Universal Robots URScript: Fase5.script

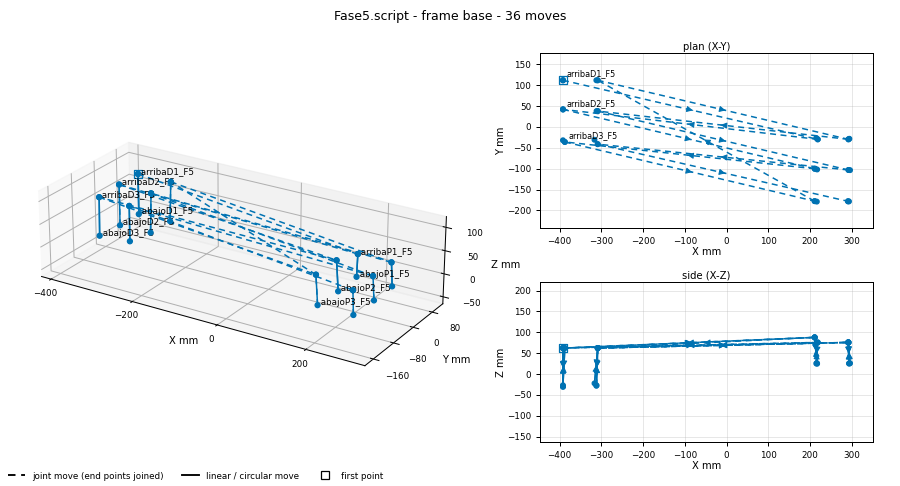
[picture p0: tool path of Fase5.script in frame base, 36 of 39 moves have a stored position in this frame; points joined in program order, loops and branches not executed]
def Fase5():
  step_count_3c5ae5f3_6041_43ff_bf36_90ec5d0922ff = 0.0
  thread Step_Counter_Thread_5067f2b5_ec87_46cd_b1bd_ecc09904e503():
    while (True):
      step_count_3c5ae5f3_6041_43ff_bf36_90ec5d0922ff = step_count_3c5ae5f3_6041_43ff_bf36_90ec5d0922ff + 1.0
      sync()
    end
  end
  run Step_Counter_Thread_5067f2b5_ec87_46cd_b1bd_ecc09904e503()
  set_standard_analog_input_domain(0, 1)
  set_standard_analog_input_domain(1, 1)
  set_tool_analog_input_domain(0, 1)
  set_tool_analog_input_domain(1, 1)
  set_analog_outputdomain(0, 0)
  set_analog_outputdomain(1, 0)
  set_input_actions_to_default()
  set_tool_communication(True, 1000000, 2, 1, 1.5, 3.5)
  set_tool_output_mode(0)
  set_tool_digital_output_mode(0, 1)
  set_tool_digital_output_mode(1, 1)
  set_tool_voltage(0)
  set_gravity([0.0, 0.0, 9.82])
  set_safety_mode_transition_hardness(1)
  set_tcp(p[0.00755148296704608,0.003639298738154023,0.026409592411711,0.0,0.0,0.0])
  set_payload(1.14, [0.022, -0.007, 0.054])
  global Mesa=p[-0.3283222416297581,-0.20095078680444134,-0.01154506462095492,-2.1087277613487028,-2.3273776320839428,-7.166709239352482E-4]
  # begin: URCap Installation Node
  #   Source: Remote TCP & Toolpath, 1.2.65.build36, Universal Robots A/S
  #   Type: Remote TCP & Toolpath
  # end: URCap Installation Node
  # begin: URCap Installation Node
  #   Source: OnRobot, 5.1.6, OnRobot A/S
  #   Type: Configuración de OnRobot
  on_robot_type = 3
  on_robot_cycle = 2.0
  on_device_ip = "localhost"
  on_device_socket_port = 51234
  on_xmlrpc = rpc_factory("xmlrpc", "http://localhost:41414")
  on_RPC = rpc_factory("xmlrpc", "http://127.0.0.1:31416")
  ON_DEBUG_LOG = False
  on_isMetric = True
  on_toolConnector = True
  on_ioqc = False
  on_dual = False
  on_ft = False
  on_hex = False
  on_gecko = 0
  on_gripper = [False, False, False]
  #======    OnRobot Globals    ======#

  ON_MATH_PI=3.141593
  ON_ZEROPOSE=p[0.0,0.0,0.0,0.0,0.0,0.0]
  ON_ZEROFRAME=p[0.0,0.0,0.0,0.0,0.0,0.0]
  ON_ZERO3D=[0.0,0.0,0.0]
  ON_ZERO6D=[0.0,0.0,0.0,0.0,0.0,0.0]
  ON_ZERO8D=[0.0,0.0,0.0,0.0,0.0,0.0,0.0,0.0]
  ON_FALSE3D=[False,False,False]
  ON_FALSE6D=[False,False,False,False,False,False]
  ON_FALSE8D=[False,False,False,False,False,False,False,False]
  global on_return=0
  on_speedL=ON_ZERO6D
  on_speedBase=ON_ZERO6D
  on_speedVect=ON_ZERO6D
  on_speedExtra=ON_ZERO6D
  on_speedDC=ON_ZERO6D
  on_speedGecko=ON_ZERO6D
  on_floatRegShift=24
  on_intRegShift=24
  on_boolRegShift=64
  ON_BASE_SHIFT_FLOAT=24
  ON_BASE_SHIFT_INT=24
  ON_BASE_SHIFT_BOOL=64
  ON_DEVICE_SHIFT_FLOAT=3
  ON_DEVICE_SHIFT_INT=2
  ON_DEVICE_SHIFT_BOOL=7
  ON_COMMON_SHIFT_FLOAT=12
  ON_COMMON_SHIFT_INT=3
  ON_COMMON_SHIFT_BOOL=1
  ON_DI_SINGLE=0
  ON_DI_PRIMARY=1
  ON_DI_SECONDARY=2
  ON_DI_DUAL=3
  ON_DEVICE_ID_MISSING=0
  ON_INIT_TIMEOUT=500
  on_robot_TCP_offset=ON_ZEROFRAME
  on_tcp_offset_actual=ON_ZEROFRAME
  on_cog_actual=ON_ZEROFRAME
  on_mass_actual=0.0
  on_robot_mount=[0.0,0.0]

  #======    End of OnRobot Globals    ======#
  #======    OnRobot Interface Messages    ======#

  on_devices_primary_log="Dispositivos de OnRobot"
  on_devices_secondary_log="Dispositivo secundario de OnRobot"
  on_device_error_title="OnRobot - Error de dispositivo"
  on_install_error="La configuración de OnRobot no es correcta.<br>Compruebe el estado en la página de configuración de OnRobot, en la pestaña de instalación.<br>Programa detenido."
  on_device_missing="No hay ningún dispositivo conectado.<br>Programa detenido."
  ft_device_missing="No hay ningún sensor F/T OnRobot conectado.<br>Programa detenido."
  rg2ft_device_missing="No hay ninguna pinza RG2-FT conectada.<br>Programa detenido."
  rg_device_missing="No hay ninguna pinza RG conectada.<br>Programa detenido."
  vg_device_missing="No hay ninguna pinza VG conectada.<br>Programa detenido."
  gg_device_missing="No hay ninguna Gecko Gripper conectada.<br>Programa detenido."
  sg_device_missing="No hay ninguna Soft Gripper conectada.<br>Programa detenido."
  tfg_device_missing="No hay ninguna pinza 3FG conectada.<br>Programa detenido."
  on_xmlrpc_start_ip="Conexión al servidor XML-RPC de OnRobot:"
  on_java_comm_error_textmsg_title="OnRobot - Error de comunicación:"
  on_java_comm_controlsocket_open_error="Apertura de la toma 'javaSocket' incorrecta."
  on_java_comm_error_title="OnRobot - Error de comunicación"
  on_java_comm_socket_open_error="El establecimiento de la conexión con el URCap ha excedido el tiempo.<br>Compruebe el estado en la página de configuración de OnRobot, en la pestaña de instalación.<br>Programa detenido."
  on_rtde_feed_error_textmsg_title="OnRobot - Error de comunicación:"
  on_rtde_feed_open_error_textmsg="Apertura de la toma 'rtdeFeed' incorrecta."
  on_rtde_feed_error_title="OnRobot - Error de comunicación"
  on_rtde_feed_open_error="El establecimiento de la conexión con los dispositivos ha excedido el tiempo.<br>Asegúrese de que los dispositivos de OnRobot funcionen y compruebe el estado en la página de configuración de OnRobot, en la pestaña de instalación."

  #======    End of OnRobot Interface Messages    ======#
  #======    OnRobot Interface    ======#

  on_portopened_javaSocket=False
  on_rtde_feed_opened=False
  on_dataRead_running=False
  FT_SENSOR_ID_UNDEFINED=0
  FT_SENSOR_ID_UNKNOWN=1
  FT_SENSOR_ID_HEX_V1=11
  FT_SENSOR_ID_HEX_V2=12
  FT_SENSOR_ID_HEX_V3=13
  FT_SENSOR_ID_RG2FT_V0=20
  FT_SENSOR_ID_RG2FT_V1=21
  FT_SENSOR_ID_RG2FT_V2=22
  def on_error(status_flag,message,title,stop_var=False):
  if(status_flag):
  popup(message,title=title,error=True,blocking=False)
  stop_var=True
  end
  return stop_var
  end
  def on_warning(status_flag,message,title):
  if(status_flag):
  textmsg(title,message)
  end
  end
  def on_missing():
  popup(on_device_missing,title=on_device_error_title,error=True,blocking=False)
  halt
  end
  def ft_missing():
  popup(ft_device_missing,title=on_device_error_title,error=True,blocking=False)
  halt
  end
  def rg2ft_missing():
  popup(rg2ft_device_missing,title=on_device_error_title,error=True,blocking=False)
  halt
  end
  def rg_missing():
  popup(rg_device_missing,title=on_device_error_title,error=True,blocking=False)
  halt
  end
  def vg_missing():
  popup(vg_device_missing,title=on_device_error_title,error=True,blocking=False)
  halt
  end
  def gg_missing():
  popup(gg_device_missing,title=on_device_error_title,error=True,blocking=False)
  halt
  end
  def sg_missing():
  popup(sg_device_missing,title=on_device_error_title,error=True,blocking=False)
  halt
  end
  def tfg_missing():
  popup(tfg_device_missing,title=on_device_error_title,error=True,blocking=False)
  halt
  end
  def on_portclose_javaSocket():
  socket_close("javaSocket")
  on_portopened_javaSocket=False
  end
  def on_portopen_javaSocket():
  on_portclose_javaSocket()
  on_portopened_javaSocket=socket_open("127.0.0.1",44005,"javaSocket")
  if not on_portopened_javaSocket:
  textmsg(on_java_comm_error_textmsg_title,on_java_comm_controlsocket_open_error)
  popup(on_java_comm_socket_open_error,title=on_java_comm_error_title,error=True,blocking=False)
  halt
  end
  end
  def on_rtde_feed_close():
  socket_close("rtdeFeed")
  on_rtde_feed_opened=False
  end
  def on_rtde_feed_open():
  on_rtde_feed_close()
  on_rtde_feed_opened=socket_open(on_device_ip,on_device_socket_port,"rtdeFeed")
  if not on_rtde_feed_opened:
  on_rtde_feed_opened=socket_open(on_device_ip,on_device_socket_port,"rtdeFeed")
  end
  if not on_rtde_feed_opened:
  textmsg(on_rtde_feed_error_textmsg_title,on_rtde_feed_open_error_textmsg)
  popup(on_rtde_feed_open_error,title=on_rtde_feed_error_title,error=True,blocking=False)
  halt
  end
  end
  def on_dataRead():
  enter_critical
  floatRegDummy=read_input_float_register(0+on_floatRegShift)
  on_speedVect[0]=floatRegDummy/1000.0
  floatRegDummy=read_input_float_register(1+on_floatRegShift)
  on_speedVect[1]=floatRegDummy/1000.0
  floatRegDummy=read_input_float_register(2+on_floatRegShift)
  on_speedVect[2]=floatRegDummy/1000.0
  floatRegDummy=read_input_float_register(3+on_floatRegShift)
  on_speedVect[3]=floatRegDummy
  floatRegDummy=read_input_float_register(4+on_floatRegShift)
  on_speedVect[4]=floatRegDummy
  floatRegDummy=read_input_float_register(5+on_floatRegShift)
  on_speedVect[5]=floatRegDummy
  exit_critical
  end
  def on_set_rtde_watchdog(updateHz=5,ftWD=False,gripperWD=-1):
  local update_str=str_cat(" watchdog set to [Hz]: ",updateHz)
  if ftWD:
  watchdog_int_reg_str=str_cat("input_int_register_",0+on_intRegShift)
  rtde_set_watchdog(watchdog_int_reg_str,updateHz,"stop")
  if ON_DEBUG_LOG:
  textmsg(watchdog_int_reg_str,update_str)
  end
  end
  if not(gripperWD<0):
  if(gripperWD==ON_DI_SINGLE or gripperWD==ON_DI_PRIMARY or gripperWD==ON_DI_DUAL):
  watchdog_int_reg_str=str_cat("input_int_register_",3+on_intRegShift)
  rtde_set_watchdog(watchdog_int_reg_str,updateHz,"stop")
  if ON_DEBUG_LOG:
  textmsg(watchdog_int_reg_str,update_str)
  end
  end
  if(gripperWD==ON_DI_SECONDARY or gripperWD==ON_DI_DUAL):
  watchdog_int_reg_str=str_cat("input_int_register_",ON_DEVICE_SHIFT_INT+3+on_intRegShift)
  rtde_set_watchdog(watchdog_int_reg_str,updateHz,"stop")
  if ON_DEBUG_LOG:
  textmsg(watchdog_int_reg_str,update_str)
  end
  end
  end
  end
  def on_speedVect_get():
  return[on_speedVect[0],on_speedVect[1],on_speedVect[2],on_speedVect[3],on_speedVect[4],on_speedVect[5]]
  end
  def on_speedDC_get():
  local speedExtra=ON_ZERO6D
  if on_speedl_for_depthcompensation:
  speedExtra=[on_speedDC[0],on_speedDC[1],on_speedDC[2],on_speedDC[3],on_speedDC[4],on_speedDC[5]]
  end
  return speedExtra
  end
  def on_speedDC_set(speedDC):
  on_speedDC=[speedDC[0],speedDC[1],speedDC[2],speedDC[3],speedDC[4],speedDC[5]]
  end
  def on_speedGecko_get():
  local speedExtra=ON_ZERO6D
  if on_speedl_for_gecko:
  speedExtra=[on_speedGecko[0],on_speedGecko[1],on_speedGecko[2],on_speedGecko[3],on_speedGecko[4],on_speedGecko[5]]
  end
  return speedExtra
  end
  def on_speedGecko_set(speedGecko):
  on_speedGecko=[speedGecko[0],speedGecko[1],speedGecko[2],speedGecko[3],speedGecko[4],speedGecko[5]]
  end
  thread on_dataRead_thread():
  if ON_DEBUG_LOG:
  textmsg("Starting on_dataRead thread")
  end
  while on_dataRead_running:
  sync()
  on_dataRead()
  end
  if ON_DEBUG_LOG:
  textmsg("Stopping on_dataRead thread")
  end
  end

  #======    End of OnRobot Interface    ======#
  #======    OnRobot QC Setup Tool Connector    ======#

  def tc_setup_tool():
  if ON_DEBUG_LOG:
  textmsg("QC Setup Tool Connector start...")
  end
  set_tool_voltage(24)

  set_tool_communication(True,1000000,2,1,1.5,3.5)

  if ON_DEBUG_LOG:
  textmsg("QC Setup Tool Connector end.")
  end
  end

  #======    End of OnRobot QC Setup Tool Connector    ======#
  #======    OnRobot TCP Messages    ======#

  on_tcp_log_msg_default="OnRobot: Desplazamiento del TCP del robot establecido en:"
  on_tcp_log_msg_primary="OnRobot: Desplazamiento del TCP del robot establecido en primario:"
  on_tcp_log_msg_secondary="OnRobot: Desplazamiento del TCP del robot establecido en secundario:"

  #======    End of OnRobot TCP Messages    ======#
  #======    OnRobot TCP    ======#

  on_tcp_offset_actual=ON_ZEROFRAME
  on_tcp_offset_primary=ON_ZEROFRAME
  on_tcp_static_primary=ON_ZEROFRAME
  on_tcp_dynamic_primary=ON_ZEROFRAME
  on_tcp_vision_primary=ON_ZEROFRAME
  on_tcp_qc_primary=ON_ZEROFRAME
  on_tcp_base_primary=ON_ZEROFRAME
  on_tcp_gripper_static_primary=ON_ZEROFRAME
  on_tcp_tool_primary=ON_ZEROFRAME
  on_tcp_gripper_dynamic_primary=ON_ZEROFRAME
  on_tcp_gripper_primary=ON_ZEROFRAME
  on_tcp_offset_secondary=ON_ZEROFRAME
  on_tcp_static_secondary=ON_ZEROFRAME
  on_tcp_dynamic_secondary=ON_ZEROFRAME
  on_tcp_vision_secondary=ON_ZEROFRAME
  on_tcp_qc_secondary=ON_ZEROFRAME
  on_tcp_base_secondary=ON_ZEROFRAME
  on_tcp_gripper_static_secondary=ON_ZEROFRAME
  on_tcp_tool_secondary=ON_ZEROFRAME
  on_tcp_gripper_dynamic_secondary=ON_ZEROFRAME
  on_tcp_gripper_secondary=ON_ZEROFRAME
  def on_tcp_update_primary():
  if ON_DEBUG_LOG:
  textmsg("TCP Update Primary start..")
  end
  on_tcp_gripper_dynamic_primary=p[0.0, 0.0, 0.0, 0.0, 0.0, 0.0]
  enter_critical
  on_tcp_dynamic_primary=pose_trans(on_tcp_static_primary,on_tcp_gripper_dynamic_primary)
  on_tcp_offset_primary=pose_trans(on_tcp_dynamic_primary,on_tcp_tool_primary)
  exit_critical
  if ON_DEBUG_LOG:
  textmsg("TCP Update Primary end.")
  end
  end
  def on_tcp_init_primary():
  if ON_DEBUG_LOG:
  textmsg("TCP Init Primary start..")
  end
  enter_critical
  on_tcp_base_primary=pose_trans(on_tcp_vision_primary,on_tcp_qc_primary)
  on_tcp_static_primary=pose_trans(on_tcp_base_primary,on_tcp_gripper_static_primary)
  exit_critical
  on_tcp_update_primary()
  if ON_DEBUG_LOG:
  textmsg("TCP Init Primary end.")
  end
  end
  def on_tcp_offset_set(TCP_offset):
  if ON_DEBUG_LOG:
  textmsg("TCP Offset set started!")
  end
  on_tcp_offset_send(TCP_offset)
  if(on_follow_tcp):
  set_tcp(TCP_offset)
  end
  on_robot_TCP_offset=TCP_offset
  if ON_DEBUG_LOG:
  textmsg("TCP Offset set to: ",on_robot_TCP_offset)
  end
  end
  def on_tcp_offset_forced_set_actual(isPrimary=True):
  if(not on_follow_tcp):

  local tcp_log_msg=on_tcp_log_msg_default

  textmsg(tcp_log_msg,on_tcp_offset_actual)
  set_tcp(on_tcp_offset_actual)
  end
  end
  def on_tcp_update(isPrimary=True):
  on_tcp_update_primary()

  on_tcp_set_actual_to(isPrimary)
  end
  def on_tcp_set_actual_to(isPrimary=True):

  on_tcp_offset_actual=on_tcp_offset_primary
  if(on_follow_tcp):
  textmsg(on_tcp_log_msg_default,on_tcp_offset_actual)
  end

  on_tcp_active_is_primary=isPrimary
  on_tcp_offset_set(on_tcp_offset_actual)
  end
  def on_tcp_update_tool_primary(tool_offset):
  if ON_DEBUG_LOG:
  textmsg("TCP Update Tool Primary start..")
  end
  on_tcp_tool_primary=tool_offset
  on_tcp_update_primary()
  if ON_DEBUG_LOG:
  textmsg("TCP Update Tool Primary end.")
  end
  end
  def on_tcp_tool_rpy_get(xyz=[0.0,0.0,0.0],rpy=[0.0,0.0,0.0]):
  local rotvec=rpy2rotvec(rpy)
  local tool_offset=p[xyz[0],xyz[1],xyz[2],rotvec[0],rotvec[1],rotvec[2]]
  return tool_offset
  end

  def on_tcp_update_tool(tool_offset,tool_index=0):
  if ON_DEBUG_LOG:
  textmsg("TCP Update Tool start..")
  end
  if(tool_index!=ON_DI_SECONDARY):
  on_tcp_update_tool_primary(tool_offset)
  local isPrimary=True

  end
  on_tcp_set_actual_to(isPrimary)
  if ON_DEBUG_LOG:
  textmsg("TCP Update Tool end.")
  end
  end

  #======    End of OnRobot TCP    ======#
  #======    OnRobot Payload Messages    ======#

  on_mass_log_msg="OnRobot: Masa de la carga útil del robot establecida en:"
  on_cog_log_msg="OnRobot: Centro de gravedad de la carga útil del robot establecido en:"

  #======    End of OnRobot Payload Messages    ======#
  #======    OnRobot Payload    ======#

  on_cog_actual=ON_ZEROFRAME
  on_mass_actual=0.0
  on_cog_primary=ON_ZEROFRAME
  on_cog_L1L2_primary=ON_ZEROFRAME
  on_mass_primary=0.0
  on_mass_L1L2_primary=0.0
  on_cog_vision_primary=ON_ZEROFRAME
  on_cog_qc_primary=ON_ZEROFRAME
  on_cog_base_primary=ON_ZEROFRAME
  on_cog_gripper_primary=ON_ZEROFRAME
  on_cog_tool_primary=ON_ZEROFRAME
  on_mass_vision_primary=0.0
  on_mass_qc_primary=0.0
  on_mass_base_primary=0.0
  on_mass_gripper_primary=0.0
  on_mass_tool_primary=0.0
  on_cog_secondary=ON_ZEROFRAME
  on_mass_secondary=0.0
  on_cog_gripper_secondary=ON_ZEROFRAME
  on_mass_gripper_secondary=0.0
  on_cog_tool_secondary=ON_ZEROFRAME
  on_mass_tool_secondary=0.0
  ON_LB2KG001=0.45359237/100
  def on_payload_update_primary():
  if ON_DEBUG_LOG:
  textmsg("Payload Update Primary start..")
  end
  enter_critical
  on_mass_primary=on_mass_L1L2_primary+on_mass_tool_primary
  local massL1L2L3Ratio=on_mass_tool_primary/on_mass_primary
  local toolAbsCOG=pose_trans(on_tcp_dynamic_primary,on_cog_tool_primary)
  toolAbsCOG=p[toolAbsCOG[0],toolAbsCOG[1],toolAbsCOG[2],0.0,0.0,0.0]
  on_cog_primary=interpolate_pose(on_cog_L1L2_primary,toolAbsCOG,massL1L2L3Ratio)
  on_cog_primary=p[on_cog_primary[0],on_cog_primary[1],on_cog_primary[2],0.0,0.0,0.0]
  exit_critical
  if ON_DEBUG_LOG:
  textmsg("Payload Update Primary end.")
  end
  end
  def on_payload_init_primary():
  if ON_DEBUG_LOG:
  textmsg("Payload Init Primary start..")
  end
  enter_critical
  on_mass_base_primary=on_mass_vision_primary+on_mass_qc_primary
  local massL0L1Ratio=on_mass_qc_primary/on_mass_base_primary
  on_mass_L1L2_primary=on_mass_base_primary+on_mass_gripper_primary
  local massL1L2Ratio=on_mass_gripper_primary/on_mass_L1L2_primary
  local qcAbsCOG=pose_trans(on_tcp_vision_primary,on_cog_qc_primary)
  qcAbsCOG=p[qcAbsCOG[0],qcAbsCOG[1],qcAbsCOG[2],0.0,0.0,0.0]
  on_cog_base_primary=interpolate_pose(on_cog_vision_primary,qcAbsCOG,massL0L1Ratio)
  on_cog_base_primary=p[on_cog_base_primary[0],on_cog_base_primary[1],on_cog_base_primary[2],0.0,0.0,0.0]
  local gripperAbsCOG=pose_trans(on_tcp_base_primary,on_cog_gripper_primary)
  gripperAbsCOG=p[gripperAbsCOG[0],gripperAbsCOG[1],gripperAbsCOG[2],0.0,0.0,0.0]
  on_cog_L1L2_primary=interpolate_pose(on_cog_base_primary,gripperAbsCOG,massL1L2Ratio)
  on_cog_L1L2_primary=p[on_cog_L1L2_primary[0],on_cog_L1L2_primary[1],on_cog_L1L2_primary[2],0.0,0.0,0.0]
  exit_critical
  on_payload_update_primary()
  if ON_DEBUG_LOG:
  textmsg("Payload Init Primary end.")
  end
  end
  def on_payload_update():
  on_payload_update_primary()

  on_mass_actual =on_mass_primary
  on_cog_actual=on_cog_primary

  on_payload_set_actual()
  end
  def on_payload_set_actual():

  on_mass_actual =on_mass_primary
  on_cog_actual=on_cog_primary

  local CoG=[on_cog_actual[0],on_cog_actual[1],on_cog_actual[2]]
  on_payload_set(on_mass_actual,CoG)
  end
  def on_payload_update_tool_primary(tool_mass=0,tool_cog=[0.0,0.0,0.0]):
  if ON_DEBUG_LOG:
  textmsg("Payload Update Tool Primary start..")
  end
  on_cog_tool_primary=p[tool_cog[0],tool_cog[1],tool_cog[2],0.0,0.0,0.0]
  on_mass_tool_primary=tool_mass
  on_payload_update_primary()
  if ON_DEBUG_LOG:
  textmsg("Payload Update Tool Primary end.")
  end
  end
  def on_payload_set(mass,CoG):
  if ON_DEBUG_LOG:
  textmsg("Payload set started!")
  end
  local center_of_gravity=[CoG[0],CoG[1],CoG[2]]
  on_payload_send(center_of_gravity,mass)
  if(on_isMetric):
  local roundedMass=floor(mass*100+0.5)/100
  else:
  local roundedMass=floor(mass/ON_LB2KG001+0.5)*ON_LB2KG001
  end
  set_payload(roundedMass,center_of_gravity)
  on_mass_actual=roundedMass
  on_cog_actual=p[CoG[0],CoG[1],CoG[2],0.0,0.0,0.0]
  if ON_DEBUG_LOG:
  textmsg("Payload mass, CoG set to: ",str_cat(str_cat(mass,", "),CoG))
  end
  end

  def on_payload_update_secondary():
  end
  def on_payload_init_secondary():
  end

  def on_payload_update_tool(tool_mass,tool_cog=[0.0,0.0,0.0],tool_index=0):
  if ON_DEBUG_LOG:
  textmsg("Payload Update Tool start..")
  end
  if(tool_index!=ON_DI_SECONDARY):
  on_cog_tool_primary=p[tool_cog[0],tool_cog[1],tool_cog[2],0.0,0.0,0.0]
  on_mass_tool_primary=tool_mass
  else:
  on_cog_tool_secondary=p[tool_cog[0],tool_cog[1],tool_cog[2],0.0,0.0,0.0]
  on_mass_tool_secondary=tool_mass
  end
  on_payload_update()
  if ON_DEBUG_LOG:
  textmsg("Payload Update Tool end.")
  end
  end
  def on_payload_get_cog2tcp_tool(tool_index=0):
  if(tool_index!=ON_DI_SECONDARY):
  local cog_tool=[on_tcp_tool_primary[0],on_tcp_tool_primary[1],on_tcp_tool_primary[2]]
  else:
  local cog_tool=[on_tcp_tool_secondary[0],on_tcp_tool_secondary[1],on_tcp_tool_secondary[2]]
  end
  return cog_tool
  end

  #======    End of OnRobot Payload    ======#
  #======    OnRobot QC TCP    ======#

  onrobotmini=0

  def on_tcp_offset_send(TCP_offset):
  on_robot_TCP_offset=TCP_offset
  end
  def on_payload_send(CoG,mass):
  on_robot_payload_cog=CoG
  on_robot_payload_mass=mass
  end


  #======    End of OnRobot QC TCP    ======#
  #======    OnRobot  Speedl    ======#

  on_speedl_thread_handler=0
  on_speedl_is_enabled=False
  on_speedl_is_running=False
  on_speedl_acc=0.0
  ft_speedl_hg_caranteen_reached=False
  ft_speedl_hg_caranteen_safemode=False
  on_speedl_for_ftcontrol=False
  on_speedl_for_move=False
  on_speedl_for_handguide=False
  on_speedl_for_insertpart=False
  on_speedl_for_depthcompensation=False
  on_speedl_for_center=False
  on_speedl_for_gecko=False
  on_speedl_acc=10000.0
  on_speedl_acc_to_zero=3.0
  ON_SPEEDL_FTCONTROL=1
  ON_SPEEDL_HANDGUIDE=2
  ON_SPEEDL_MOVE=3
  ON_SPEEDL_INSERTPART=4
  ON_SPEEDL_DEPTHCOMP=5
  ON_SPEEDL_CENTER=6
  ON_SPEEDL_GECKO=7
  def on_speedl_add_extra(speedBase,speedExtra):
  speedSum=ON_ZERO6D
  speedBaseP=p[speedBase[0],speedBase[1],speedBase[2],speedBase[3],speedBase[4],speedBase[5]]
  speedExtraP=p[speedExtra[0],speedExtra[1],speedExtra[2],speedExtra[3],speedExtra[4],speedExtra[5]]
  speedSumP=pose_add(speedExtraP,speedBaseP)
  speedSum=[speedSumP[0],speedSumP[1],speedSumP[2],speedSumP[3],speedSumP[4],speedSumP[5]]
  return speedSum
  end

  thread on_speedl_thread():
  if ON_DEBUG_LOG:
  textmsg("Speedl thread started..")
  end
  enter_critical
  on_speedl_is_running=True
  on_speedl_is_enabled=True
  exit_critical
  on_speedL=ON_ZERO6D

  while on_speedl_is_running:
  on_speedBase=on_speedVect_get()
  on_speedL=on_speedBase



  if on_speedl_is_enabled:
  speedl(on_speedL,a=on_speedl_acc,t=0.001)
  else:
  speedl(ON_ZERO6D,a=on_speedl_acc_to_zero,t=0.001)
  end
  end

  on_speedL=ON_ZERO6D
  if ON_DEBUG_LOG:
  textmsg("Speedl thread ended.")
  end
  end
  def on_speedl_integer_get():
  local speedl_integer=binary_list_to_integer([on_speedl_for_ftcontrol,on_speedl_for_handguide,on_speedl_for_move,on_speedl_for_insertpart,on_speedl_for_depthcompensation,on_speedl_for_center,on_speedl_for_gecko])
  return speedl_integer
  end
  def on_speedl_start_for(speedl_id):
  if(speedl_id==ON_SPEEDL_FTCONTROL):
  on_speedl_for_ftcontrol=True
  elif(speedl_id==ON_SPEEDL_HANDGUIDE):
  on_speedl_for_handguide=True
  elif(speedl_id==ON_SPEEDL_MOVE):
  on_speedl_for_move=True
  elif(speedl_id==ON_SPEEDL_INSERTPART):
  on_speedl_for_insertpart=True
  elif(speedl_id==ON_SPEEDL_DEPTHCOMP):
  on_speedl_for_depthcompensation=True
  elif(speedl_id==ON_SPEEDL_CENTER):
  on_speedl_for_center=True
  elif(speedl_id==ON_SPEEDL_GECKO):
  on_speedl_for_gecko=True
  else:
  textmsg("Unknown Start speedl ID received: ",speedl_id)
  end
  local speedl_integer=on_speedl_integer_get()
  if not(speedl_integer==0):
  if not on_speedl_is_running:
  on_speedl_thread_handler=run on_speedl_thread()
  end
  end
  return on_speedl_is_running
  end
  def on_speedl_stop_for(speedl_id,brake=10):
  if(speedl_id==ON_SPEEDL_FTCONTROL):
  on_speedl_for_ftcontrol=False
  elif(speedl_id==ON_SPEEDL_HANDGUIDE):
  on_speedl_for_handguide=False
  elif(speedl_id==ON_SPEEDL_MOVE):
  on_speedl_for_move=False
  elif(speedl_id==ON_SPEEDL_INSERTPART):
  on_speedl_for_insertpart=False
  elif(speedl_id==ON_SPEEDL_DEPTHCOMP):
  on_speedl_for_depthcompensation=False
  on_speedDC_set(ON_ZERO6D)
  elif(speedl_id==ON_SPEEDL_CENTER):
  on_speedl_for_center=False
  elif(speedl_id==ON_SPEEDL_GECKO):
  on_speedl_for_gecko=False
  on_speedGecko_set(ON_ZERO6D)
  else:
  textmsg("Unknown Stop speedl ID received: ",speedl_id)
  end
  local speedl_integer=on_speedl_integer_get()
  if(speedl_integer==0):
  if(on_speedl_is_running):
  kill on_speedl_thread_handler
  enter_critical
  on_speedl_is_running=False
  exit_critical

  end
  if ON_DEBUG_LOG:
  textmsg("Speedl thread stopped")
  end
  stopl(brake)
  end
  return on_speedl_is_running
  end
  def on_speedl_pause():
  on_speedl_is_enabled=False
  return on_speedl_integer_get()
  end
  def on_speedl_resume():
  on_speedl_is_enabled=True
  return on_speedl_integer_get()
  end
  def on_wait_ms(time_ms):
  local sync_time=ceil(norm(time_ms/2.0))
  while(sync_time>0):
  sync_time=sync_time-1
  sync()
  end
  end

  #======    End of OnRobot  Speedl    ======#
  on_install_tcp = False
  on_follow_tcp = False
  textmsg(on_devices_primary_log, ": Quick Changer + Lado de la herramienta de QC + [0.0, 0.0, 0.0, 0.0, 0.0, 0.0]")
  on_tcp_active_is_primary = True
  on_tcp_vision_primary = p[0.0, 0.0, 0.0, 0.0, 0.0, 0.0]
  on_cog_vision_primary = p[0.0, 0.0, 0.0, 0.0, 0.0, 0.0]
  on_mass_vision_primary = 0.0
  on_tcp_qc_primary = p[0.0, 0.0, 0.0136, 0.0, 0.0, 0.0]
  on_cog_qc_primary = p[0.0, 0.0, 0.004, 0.0, 0.0, 0.0]
  on_mass_qc_primary = 0.06
  on_tcp_gripper_static_primary = p[0.0, 0.0, 0.017, 0.0, 0.0, 0.0]
  on_cog_gripper_primary = p[0.0, 0.0, 0.002, 0.0, 0.0, 0.0]
  on_mass_gripper_primary = 0.14
  on_tcp_tool_primary = p[0.0, 0.0, 0.0, 0.0, 0.0, 0.0]
  on_cog_tool_primary = p[0.0, 0.0, 0.0, 0.0, 0.0, 0.0]
  on_mass_tool_primary = 0.0
  #======    OnRobot Run    ======#

  textmsg(on_xmlrpc_start_ip,on_device_ip)
  on_portopen_javaSocket()
  sync()
  on_rtde_feed_open()
  sync()
  local gripperWDs=binary_list_to_integer(on_gripper)
  if gripperWDs==0:
  gripperWDs=-1
  else:
  gripperWDs=floor(gripperWDs/2)
  end
  on_set_rtde_watchdog(updateHz=0.2,ftWD=on_ft,gripperWD=gripperWDs)
  sync()
  on_dataRead_running=True
  sync()
  on_dataRead_thrd=run on_dataRead_thread()
  sync()
  on_tcp_init_primary()
  on_payload_init_primary()

  on_tcp_set_actual_to(on_tcp_active_is_primary)
  if(on_follow_tcp):
  on_payload_set_actual()
  end

  #======    End of OnRobot Run    ======#
  #======    OnRobot QC Start    ======#

  if(on_toolConnector):
  tc_setup_tool()
  end
  sync()

  #======    End of OnRobot QC Start    ======#
  # end: URCap Installation Node
  global arribaD1_F5_p=p[-.391906112680, .111701728632, .062414730639, -3.120840940537, -.027823823919, .013083639781]
  global arribaD1_F5_q=[-0.5999215284930379, -1.2160912317088552, 1.347379032765519, -1.7217775783934712, -1.5846818129169158, 0.957253456115742]
  global abajoD1_F5_p=p[-.391903107168, .111738401018, -.030076558729, -3.120770850857, -.027780336222, .013081599309]
  global abajoD1_F5_q=[-0.5994060675250292, -1.09217269838366, 1.6244571844683948, -2.122820039788717, -1.5855448881732581, 0.9567382335662976]
  global arribaP1_F5_p=p[.218348772489, -.029777054927, .075818997484, -2.208073880386, -2.214622291990, .011868549599]
  global arribaP1_F5_q=[0.4763003528692451, -1.0782644118820848, -2.0530307991209398, -1.591565744893618, 1.5791739072044746, -2.664245103169357]
  global abajoP1_F5_p=p[.214883970739, -.026553408258, .025332433947, -2.208096720401, -2.214564325806, .012029326262]
  global abajoP1_F5_q=[0.5012585611728304, -1.0828022679372111, -2.289871978616599, -1.350012176417624, 1.5798720389052319, -2.639810493641351]
  global arribaD2_F5_p=p[-.391905729757, .041937664632, .062414616985, -3.120852674643, -.027796367923, .013097560852]
  global arribaD2_F5_q=[-0.4378894011127308, -1.2707415384105225, 1.421295468007215, -1.7388397655882502, -1.5872953573809507, 1.119180917739829]
  global abajoD2_F5_p=p[-.391925924350, .041973913384, -.030436105952, -3.120816661988, -.027707776863, .013220657936]
  global abajoD2_F5_q=[-0.43733865419502926, -1.1382590097240133, 1.698486153279445, -2.1486069164671457, -1.5881102720842977, 1.1187369823455224]
  global arribaP2_F5_p=p[.211131703305, -.100237661043, .087809202549, -2.207719815606, -2.214325776079, .012411491345]
  global arribaP2_F5_q=[0.13561208287999155, -1.153139036792644, -1.9579103548872432, -1.6154767556459637, 1.574461518224063, -3.004933373158606]
  global abajoP2_F5_p=p[.216857083786, -.101946153601, .024825938304, -2.207758626392, -2.214496629550, .012426880076]
  global abajoP2_F5_q=[0.12409290981682985, -1.2259192666008545, -2.2158700183319615, -1.2847368623930713, 1.5744615182240613, -3.017325210847757]
  global arribaD3_F5_p=p[-.387504120003, -.036086832394, .062415367671, -3.120876650693, -.027762251239, .013123928534]
  global arribaD3_F5_q=[-0.24047118822208802, -1.2873407167247422, 1.4420540968524511, -1.7397476635375, -1.5901244322405947, 1.3165955543517764]
  global abajoD3_F5_p=p[-.391986462235, -.032023567276, -.026846823760, -3.120886510452, -.027672463694, .013026002921]
  global abajoD3_F5_q=[-0.24771434465520592, -1.1455655854991589, 1.6885622183429332, -2.128113885919083, -1.5908797422991743, 1.3084404468536015]
  global arribaP3_F5_p=p[.210893817940, -.177854700257, .087997554369, -2.188403404214, -2.233894388107, .010988382706]
  global arribaP3_F5_q=[-0.21223203704250793, -1.361705882405964, -1.8210765415308963, -1.5444418550897723, 1.568527398767303, -3.370754384376644]
  global abajoP3_F5_p=p[.216105806086, -.178974782601, .026430992677, -2.198642191659, -2.243980104786, -.003370439817]
  global abajoP3_F5_q=[-0.2122429052611272, -1.4184752267232525, -2.0787739754150465, -1.2129412454205646, 1.5689954757415014, -3.3714225927542576]
  global arribaD4_F5_p=p[-.308728627987, .111696866569, .062402999374, -3.120867802786, -.027806215010, .012992685041]
  global arribaD4_F5_q=[-0.7530906836139284, -1.5632954400828725, 1.7666180769549573, -1.7954021892943075, -1.5803898016558877, 0.8033258914947377]
  global abajoD4_F5_p=p[-.311996402408, .111703062929, -.027985996874, -3.120815093988, -.027892998692, .013125268678]
  global abajoD4_F5_q=[-0.7447097937213778, -1.387084321384748, 2.0390918890581933, -2.2441145382322256, -1.5813849608050212, 0.8107097148894733]
  global arribaP4_F5_p=p[.291895942277, -.029765667268, .075842881749, -2.210018597693, -2.212578570616, .011566612677]
  global arribaP4_F5_q=[0.346447856520875, -1.4498450096317193, -1.8078120392156904, -1.466425637525667, 1.5763813804012772, -2.793050401966526]
  global abajoP4_F5_p=p[.294119413153, -.028411347682, .025236657727, -2.209935310745, -2.212601920624, .011559542046]
  global abajoP4_F5_q=[0.34836771869812305, -1.5125023297782372, -1.9968311972067632, -1.214749159388031, 1.5767304462516272, -2.7918286714900793]
  global arribaD5_F5_p=p[-.308723734132, .037870064631, .062393292850, -3.120905149481, -.027819638057, .012956496600]
  global arribaD5_F5_q=[-0.5477364698992613, -1.6365057430663263, 1.8362644354450075, -1.7894998989501545, -1.5840223471271457, 1.0084681510925781]
  global abajoD5_F5_p=p[-.311560454526, .037877309669, -.026954983583, -3.120879399455, -.027842728673, .013015518749]
  global abajoD5_F5_q=[-0.5414508024799023, -1.4573550981334424, 2.11683637300602, -2.2491961918272807, -1.5849698225604012, 1.0138242244720184]
  global arribaP5_F5_p=p[.292047162969, -.103183589286, .075859924159, -2.208132210748, -2.214600453443, .011672001046]
  global arribaP5_F5_q=[0.08726646259972791, -1.5250687003925991, -1.7386970008368081, -1.462411380246003, 1.5723671231216807, -3.054151658064867]
  global abajoP5_F5_p=p[.295705794105, -.103593395841, .026035264610, -2.208122401487, -2.214676175333, .011698322582]
  global abajoP5_F5_q=[0.0848230016469224, -1.592438409519608, -1.9135789918866095, -1.2201596800692096, 1.5725416560468926, -3.057293250718453]
  global arribaD6_F5_p=p[-.308718960545, -.041374722305, .062384791718, -3.120903917091, -.027837002597, .012928111769]
  global arribaD6_F5_q=[-0.28755122820006385, -1.6276790104308096, 1.8264959494220296, -1.7845674953856658, -1.5882065931903568, 1.268661737442052]
  global abajoD6_F5_p=p[-.316426570259, -.030792570349, -.022202075799, -3.090293169514, -.025741052345, .110028741673]
  global abajoD6_F5_q=[-0.3058436552631072, -1.5009167951396591, 2.1768983046161186, -2.330723424951067, -1.5966704527484081, 1.2494904994964324]
  global arribaP6_F6_p=p[.290842154195, -.178201610540, .075861425338, -2.208296211563, -2.214456686254, .011699172526]
  global arribaP6_F6_q=[-0.1603957582582467, -1.6639969088513293, -1.5952309363229054, -1.4679964338523668, 1.5680037999916725, -3.3019884118480434]
  global abajoP6_F5_p=p[.293146068160, -.178483438405, .025420318775, -2.208421334940, -2.214288626345, .011635200503]
  global abajoP6_F5_q=[-0.1602212253330908, -1.7221163729428781, -1.7725563883253317, -1.2325515177584982, 1.568352865842117, -3.302337477698492]
  $ 1 "Programa de robot"
  $ 2 "'Program generated by RoboDK v5.2.2 for UR3e on 10/11/2021 09:56:11'"
  # 'Program generated by RoboDK v5.2.2 for UR3e on 10/11/2021 09:56:11'
  $ 3 "'Using nominal kinematics.'"
  # 'Using nominal kinematics.'
  $ 4 "'Using Ref. PosicionD: p[0.161767, -0.119777, -0.855711, -0.000000, 0.000000, 3.141593]'"
  # 'Using Ref. PosicionD: p[0.161767, -0.119777, -0.855711, -0.000000, 0.000000, 3.141593]'
  $ 5 "Ajustar DO[1]=Apagar"
  set_standard_digital_out(1, False)
  $ 6 "i≔1"
  global i=1
  $ 7 "Inicio"
  movej([0.0, -1.5707963267948966, 0.0, -1.5707963267948966, 0.0, 0.0], a=1.3962634015954636, v=1.0471975511965976)
  $ 8 "'Using TCP SAI6199-GV_E1_jt: p[0.000000, 0.000000, 0.200000, 0.000000, 0.000000, 0.000000]'"
  # 'Using TCP SAI6199-GV_E1_jt: p[0.000000, 0.000000, 0.200000, 0.000000, 0.000000, 0.000000]'
  $ 9 "set_tcp(p[0.000000, 0.000000, 0.200000, 0.000000, 0.000000, 0.000000])"
  set_tcp(p[0.000000, 0.000000, 0.200000, 0.000000, 0.000000, 0.000000])
  $ 10 "Bucle i≤6"
  while (i <= 6):
    $ 12 "If i≟1"
    if (i == 1):
      $ 13 "MoverJ"
      $ 14 "arribaD1_F5" "breakAfter"
      movej(get_inverse_kin(arribaD1_F5_p, qnear=arribaD1_F5_q), a=1.3962634015954636, v=1.0471975511965976)
      $ 15 "MoverL"
      $ 16 "abajoD1_F5" "breakAfter"
      movel(abajoD1_F5_p, a=1.2, v=0.25)
      $ 17 "Esperar: 0.5"
      sleep(0.5)
      $ 18 "Ajustar DO[1]=Encender"
      set_standard_digital_out(1, True)
      $ 19 "Esperar: 0.5"
      sleep(0.5)
      $ 20 "MoverL"
      $ 21 "arribaD1_F5" "breakAfter"
      movel(arribaD1_F5_p, a=1.2, v=0.25)
      $ 22 "MoverJ"
      $ 23 "arribaP1_F5" "breakAfter"
      movej(get_inverse_kin(arribaP1_F5_p, qnear=arribaP1_F5_q), a=1.3962634015954636, v=1.0471975511965976)
      $ 24 "MoverL"
      $ 25 "abajoP1_F5" "breakAfter"
      movel(abajoP1_F5_p, a=1.2, v=0.25)
      $ 26 "Esperar: 0.5"
      sleep(0.5)
      $ 27 "Ajustar DO[1]=Apagar"
      set_standard_digital_out(1, False)
      $ 28 "Esperar: 0.5"
      sleep(0.5)
      $ 29 "MoverL"
      $ 30 "arribaP1_F5" "breakAfter"
      movel(arribaP1_F5_p, a=1.2, v=0.25)
    else:
      $ 31 "ElseIf i≟2"
      if (i == 2):
        $ 32 "MoverJ"
        $ 33 "arribaD2_F5" "breakAfter"
        movej(get_inverse_kin(arribaD2_F5_p, qnear=arribaD2_F5_q), a=1.3962634015954636, v=1.0471975511965976)
        $ 34 "MoverL"
        $ 35 "abajoD2_F5" "breakAfter"
        movel(abajoD2_F5_p, a=1.2, v=0.25)
        $ 36 "Esperar: 0.5"
        sleep(0.5)
        $ 37 "Ajustar DO[1]=Encender"
        set_standard_digital_out(1, True)
        $ 38 "Esperar: 0.5"
        sleep(0.5)
        $ 39 "MoverJ"
        $ 40 "arribaD2_F5" "breakAfter"
        movej(get_inverse_kin(arribaD2_F5_p, qnear=arribaD2_F5_q), a=1.3962634015954636, v=1.0471975511965976)
        $ 41 "arribaP2_F5" "breakAfter"
        movej(get_inverse_kin(arribaP2_F5_p, qnear=arribaP2_F5_q), a=1.3962634015954636, v=1.0471975511965976)
        $ 42 "MoverL"
        $ 43 "abajoP2_F5" "breakAfter"
        movel(abajoP2_F5_p, a=1.2, v=0.25)
        $ 44 "Esperar: 0.5"
        sleep(0.5)
        $ 45 "Ajustar DO[1]=Apagar"
        set_standard_digital_out(1, False)
        $ 46 "Esperar: 0.5"
        sleep(0.5)
        $ 47 "MoverL"
        $ 48 "arribaP2_F5" "breakAfter"
        movel(arribaP2_F5_p, a=1.2, v=0.25)
      else:
        $ 49 "ElseIf i≟3"
        if (i == 3):
          $ 50 "MoverJ"
          $ 51 "arribaD3_F5" "breakAfter"
          movej(get_inverse_kin(arribaD3_F5_p, qnear=arribaD3_F5_q), a=1.3962634015954636, v=1.0471975511965976)
          $ 52 "MoverL"
          $ 53 "abajoD3_F5" "breakAfter"
          movel(abajoD3_F5_p, a=1.2, v=0.25)
          $ 54 "Esperar: 0.5"
          sleep(0.5)
          $ 55 "Ajustar DO[1]=Encender"
          set_standard_digital_out(1, True)
          $ 56 "Esperar: 0.5"
          sleep(0.5)
          $ 57 "MoverL"
          $ 58 "arribaD3_F5" "breakAfter"
          movel(arribaD3_F5_p, a=1.2, v=0.25)
          $ 59 "MoverJ"
          $ 60 "arribaP3_F5" "breakAfter"
          movej(get_inverse_kin(arribaP3_F5_p, qnear=arribaP3_F5_q), a=1.3962634015954636, v=1.0471975511965976)
          $ 61 "MoverL"
          $ 62 "abajoP3_F5" "breakAfter"
          movel(abajoP3_F5_p, a=1.2, v=0.25)
          $ 63 "Esperar: 0.5"
          sleep(0.5)
          $ 64 "Ajustar DO[1]=Apagar"
          set_standard_digital_out(1, False)
          $ 65 "Esperar: 0.5"
          sleep(0.5)
          $ 66 "MoverJ"
          $ 67 "arribaP3_F5" "breakAfter"
          movej(get_inverse_kin(arribaP3_F5_p, qnear=arribaP3_F5_q), a=1.3962634015954636, v=1.0471975511965976)
        else:
          $ 68 "ElseIf i≟4"
          if (i == 4):
            $ 69 "MoverJ"
            $ 70 "arribaD4_F5" "breakAfter"
            movej(get_inverse_kin(arribaD4_F5_p, qnear=arribaD4_F5_q), a=1.3962634015954636, v=1.0471975511965976)
            $ 71 "MoverL"
            $ 72 "abajoD4_F5" "breakAfter"
            movel(abajoD4_F5_p, a=1.2, v=0.25)
            $ 73 "Esperar: 0.5"
            sleep(0.5)
            $ 74 "Ajustar DO[1]=Encender"
            set_standard_digital_out(1, True)
            $ 75 "Esperar: 0.5"
            sleep(0.5)
            $ 76 "MoverJ"
            $ 77 "arribaD4_F5" "breakAfter"
            movej(get_inverse_kin(arribaD4_F5_p, qnear=arribaD4_F5_q), a=1.3962634015954636, v=1.0471975511965976)
            $ 78 "MoverJ"
            $ 79 "arribaP4_F5" "breakAfter"
            movej(get_inverse_kin(arribaP4_F5_p, qnear=arribaP4_F5_q), a=1.3962634015954636, v=1.0471975511965976)
            $ 80 "MoverL"
            $ 81 "abajoP4_F5" "breakAfter"
            movel(abajoP4_F5_p, a=1.2, v=0.25)
            $ 82 "Esperar: 0.5"
            sleep(0.5)
            $ 83 "Ajustar DO[1]=Apagar"
            set_standard_digital_out(1, False)
            $ 84 "Esperar: 0.5"
            sleep(0.5)
            $ 85 "MoverL"
            $ 86 "arribaP4_F5" "breakAfter"
            movel(arribaP4_F5_p, a=1.2, v=0.25)
          else:
            $ 87 "ElseIf i≟5"
            if (i == 5):
              $ 88 "MoverJ"
              $ 89 "arribaD5_F5" "breakAfter"
              movej(get_inverse_kin(arribaD5_F5_p, qnear=arribaD5_F5_q), a=1.3962634015954636, v=1.0471975511965976)
              $ 90 "MoverJ"
              $ 91 "abajoD5_F5" "breakAfter"
              movej(get_inverse_kin(abajoD5_F5_p, qnear=abajoD5_F5_q), a=1.3962634015954636, v=1.0471975511965976)
              $ 92 "Esperar: 0.5"
              sleep(0.5)
              $ 93 "Ajustar DO[1]=Encender"
              set_standard_digital_out(1, True)
              $ 94 "Esperar: 0.5"
              sleep(0.5)
              $ 95 "MoverL"
              $ 96 "arribaD5_F5" "breakAfter"
              movel(arribaD5_F5_p, a=1.2, v=0.25)
              $ 97 "MoverJ"
              $ 98 "arribaP5_F5" "breakAfter"
              movej(get_inverse_kin(arribaP5_F5_p, qnear=arribaP5_F5_q), a=1.3962634015954636, v=1.0471975511965976)
              $ 99 "MoverL"
              $ 100 "abajoP5_F5" "breakAfter"
              movel(abajoP5_F5_p, a=1.2, v=0.25)
              $ 101 "Esperar: 0.5"
              sleep(0.5)
              $ 102 "Ajustar DO[1]=Apagar"
              set_standard_digital_out(1, False)
              $ 103 "Esperar: 0.5"
              sleep(0.5)
              $ 104 "MoverJ"
              $ 105 "arribaP5_F5" "breakAfter"
              movej(get_inverse_kin(arribaP5_F5_p, qnear=arribaP5_F5_q), a=1.3962634015954636, v=1.0471975511965976)
            else:
              $ 106 "ElseIf i≟6"
              if (i == 6):
                $ 107 "MoverJ"
                $ 108 "arribaD6_F5" "breakAfter"
                movej(get_inverse_kin(arribaD6_F5_p, qnear=arribaD6_F5_q), a=1.3962634015954636, v=1.0471975511965976)
                $ 109 "MoverL"
                $ 110 "abajoD6_F5" "breakAfter"
                movel(abajoD6_F5_p, a=1.2, v=0.25)
                $ 111 "Esperar: 0.5"
                sleep(0.5)
                $ 112 "Ajustar DO[1]=Encender"
                set_standard_digital_out(1, True)
                $ 113 "Esperar: 0.5"
                sleep(0.5)
                $ 114 "MoverL"
                $ 115 "arribaD6_F5" "breakAfter"
                movel(arribaD6_F5_p, a=1.2, v=0.25)
                $ 116 "MoverJ"
                $ 117 "arribaP6_F6" "breakAfter"
                movej(get_inverse_kin(arribaP6_F6_p, qnear=arribaP6_F6_q), a=1.3962634015954636, v=1.0471975511965976)
                $ 118 "MoverL"
                $ 119 "abajoP6_F5" "breakAfter"
                movel(abajoP6_F5_p, a=1.2, v=0.25)
                $ 120 "Esperar: 0.5"
                sleep(0.5)
                $ 121 "Ajustar DO[1]=Apagar"
                set_standard_digital_out(1, False)
                $ 122 "Esperar: 0.5"
                sleep(0.5)
                $ 123 "MoverJ"
                $ 124 "arribaP6_F6" "breakAfter"
                movej(get_inverse_kin(arribaP6_F6_p, qnear=arribaP6_F6_q), a=1.3962634015954636, v=1.0471975511965976)
              end
            end
          end
        end
      end
    end
    $ 125 "NumPiezas≔i"
    global NumPiezas=i
    $ 126 "i≔i+1"
    global i=i+1
  end
  $ 127 "movej([0.017453, -1.553343, 0.017453, -1.553343, 0.017453, 0.017453],1.20000,0.25000,0,0.0000)"
  movej([0.017453, -1.553343, 0.017453, -1.553343, 0.017453, 0.017453],1.20000,0.25000,0,0.0000)
  $ 128 "Inicio"
  movej([0.0, -1.5707963267948966, 0.0, -1.5707963267948966, 0.0, 0.0], a=1.3962634015954636, v=1.0471975511965976)
end
